// TIA Portal V20 export
TYPE "Buttons"
   STRUCT
      Start : Bool;
      Stop : Bool;
      Reset : Bool;
      "Emergency stop" : Bool;
   END_STRUCT;
END_TYPE
